(* PLC project gray_encoder, Dassault Systèmes ControlBuild 2024x *)
(* stored: creationDateTime 2023-10-03T11:12:51-01:00 *)

(* This module simulates the behaviour of a Gray encoder. *)
FUNCTION_BLOCK equipment_library.gray_encoder
  VAR_INPUT
    binaryInput : DINT := 0;
    encoderFreezing : BOOL := false;
  END_VAR
  VAR_OUTPUT
    bit00 : BOOL := false;
    bit01 : BOOL := false;
    bit02 : BOOL := false;
    bit03 : BOOL := false;
    bit04 : BOOL := false;
    bit05 : BOOL := false;
    bit06 : BOOL := false;
    bit07 : BOOL := false;
    bit08 : BOOL := false;
    bit09 : BOOL := false;
    bit10 : BOOL := false;
    bit11 : BOOL := false;
    bit12 : BOOL := false;
    bit13 : BOOL := false;
    bit14 : BOOL := false;
    bit15 : BOOL := false;
    wordOutput : DINT := 0;
  END_VAR
  VAR
    validBit : BOOL := false;
    testValue : DINT := 0;
    index : DINT := 0;
    rank : REAL := 0.0;
    memoRank : DINT := 0;
    inputValue : DINT := 0;
  END_VAR
  VAR
    d_presetting : BOOL := false;
    v_d_presetting : DINT := 0;
  END_VAR


ACTION C_source_code:
/* ----------------------------------------------------------------	*/
/* Type : Model of Operative Behaviour					*/
/* Category :  Sensors							*/
/* Author : Dassault Systemes						*/
/* Update date : June 2018							*/
/* ----------------------------------------------------------------	*/
/* This module simulates the behaviour 					*/
/*   of a Gray encoder							*/ 
/* ----------------------------------------------------------------	*/
/* ----------------------------------------------------------------	*/
/* Treatment of presetting fault						*/
/* ----------------------------------------------------------------	*/
if (d_presetting) inputValue = v_d_presetting;
else inputValue = binaryInput;


/* ----------------------------------------------------------------	*/
/* Encoder management							*/
/* ----------------------------------------------------------------	*/
if (d_presetting) inputValue = v_d_presetting;
else inputValue = binaryInput;

if (!encoderFreezing) {
	if(inputValue < 65535) {
		wordOutput = 0;
		for (index = 0;index<=15;index++) {
			rank = pow(2.0,(2.0+index));
			memoRank = rank;
			testValue = inputValue % memoRank;
			validBit = 0;
			if (  (( rank /4) <= testValue  ) && ( testValue  < ( rank * 3 /4 ) )  ) validBit = 1;
			switch (index) {
				case 0:
					bit00 = validBit;
					if (validBit) wordOutput = wordOutput +pow(2.0,0.0);
					break;
				case 1:
					bit01 = validBit;
					if (validBit) wordOutput = wordOutput +pow(2.0,1.0);
					break;
				case 2:
					bit02 = validBit;
					if (validBit) wordOutput = wordOutput +pow(2.0,2.0);
					break;
				case 3:
					bit03 = validBit;
					if (validBit) wordOutput = wordOutput +pow(2.0,3.0);
					break;
				case 4:
					bit04 = validBit;
					if (validBit) wordOutput = wordOutput +pow(2.0,4.0);
					break;
				case 5:
					bit05 = validBit;
					if (validBit) wordOutput = wordOutput +pow(2.0,5.0);
					break;
				case 6:
					bit06 = validBit;
					if (validBit) wordOutput = wordOutput +pow(2.0,6.0);
					break;
				case 7:
					bit07 = validBit;
					if (validBit) wordOutput = wordOutput +pow(2.0,7.0);
					break;
				case 8:
					bit08 = validBit;
					if (validBit) wordOutput = wordOutput +pow(2.0,8.0);
					break;
				case 9:
					bit09 = validBit;
					if (validBit) wordOutput = wordOutput +pow(2.0,9.0);
					break;
				case 10:
					bit10 = validBit;
					if (validBit) wordOutput = wordOutput +pow(2.0,10.0);
					break;
				case 11:
					bit11 = validBit;
					if (validBit) wordOutput = wordOutput +pow(2.0,11.0);
					break;
				case 12:
					bit12 = validBit;
					if (validBit) wordOutput = wordOutput +pow(2.0,12.0);
					break;
				case 13:
					bit13 = validBit;
					if (validBit) wordOutput = wordOutput +pow(2.0,13.0);
					break;
				case 14:
					bit14 = validBit;
					if (validBit) wordOutput = wordOutput +pow(2.0,14.0);
					break;
				case 15:
					bit15 = validBit;
					if (validBit) wordOutput = wordOutput +pow(2.0,15.0);
					break;
			}
		}
	}
	else {
		bit00 = 0;
		bit01 = 0;
		bit02 = 0;
		bit03 = 0;
		bit04 = 0;
		bit05 = 0;
		bit06 = 0;
		bit07 = 0;
		bit08 = 0;
		bit09 = 0;
		bit10 = 0;
		bit11 = 0;
		bit12 = 0;
		bit13 = 0;
		bit14 = 0;
		bit15 = 0;
		wordOutput = 0;
	}
}
END_ACTION

ACTION C_header:
#include <math.h>
END_ACTION
END_FUNCTION_BLOCK
